FUNCTION_BLOCK MoveVelo IMPLEMENTS I_MoveVelo
VAR
	mcMoveVelo : MC_MoveVelocity;
END_VAR
VAR_IN_OUT
	Axis : AXIS_REF;
END_VAR

mcMoveVelo(Axis := Axis);

PROPERTY Acceleration : MC_LREAL
GET
Acceleration := mcMoveVelo.Acceleration;
END_GET
SET
mcMoveVelo.Acceleration := Acceleration;
END_SET
END_PROPERTY

PROPERTY BufferMode : MC_Buffermode
GET
BufferMode := mcMoveVelo.BufferMode;
END_GET
SET
mcMoveVelo.BufferMode := BufferMode;
END_SET
END_PROPERTY

PROPERTY Busy : BOOL
GET
Busy := mcMoveVelo.Busy;
END_GET
END_PROPERTY

PROPERTY Deceleration : MC_LREAL
GET
Deceleration := mcMoveVelo.Deceleration;
END_GET
SET
mcMoveVelo.Deceleration := Deceleration;
END_SET
END_PROPERTY

PROPERTY Direction : MC_Direction
GET
Direction := mcMoveVelo.Direction;
END_GET
SET
mcMoveVelo.Direction := Direction;
END_SET
END_PROPERTY

PROPERTY Done : BOOL
GET
Done := mcMoveVelo.Done;
END_GET
END_PROPERTY

PROPERTY Error : BOOL
GET
Error := mcMoveVelo.Error;
END_GET
END_PROPERTY

PROPERTY Execute : BOOL
GET
Execute := mcMoveVelo.Execute;
END_GET
SET
mcMoveVelo.Execute := Execute;
END_SET
END_PROPERTY

PROPERTY InVelocity : BOOL
GET
InVelocity := mcMoveVelo.InVelocity;
END_GET
END_PROPERTY

PROPERTY Jerk : MC_LREAL
GET
Jerk := mcMoveVelo.Jerk;
END_GET
SET
mcMoveVelo.Jerk := Jerk;
END_SET
END_PROPERTY

PROPERTY Velocity : MC_LREAL
GET
Velocity := mcMoveVelo.Velocity;
END_GET
SET
mcMoveVelo.Velocity := Velocity;
END_SET
END_PROPERTY

END_FUNCTION_BLOCK

(* stored: Version 1.1.0.1
   POU MoveVelo: Id {11334e21-52f4-414b-aae4-bc02cc7be0a4}, SpecialFunc None
   Property Acceleration: Id {58f1d593-40f0-476d-a5a7-9b3cb778c7d3}
   Get Get: Id {954d0383-4be7-4b14-9478-9d1fb760cc0e}
   Set Set: Id {fc4bfc0a-ae1e-4e71-8268-d6b467dad374}
   Property BufferMode: Id {acef93d6-5f3f-4775-9fbb-a2c1a4097a54}
   Get Get: Id {fc2e896c-3b8e-490c-bad6-bfe7d1ca6171}
   Set Set: Id {3885e3b8-2b10-4b89-92bf-e144af053276}
   Property Busy: Id {316065bc-29d0-4424-a035-e7821cbdb68e}
   Get Get: Id {0304dd71-866f-4d72-94c8-7ce48bc29350}
   Property Deceleration: Id {0eca7112-34e1-452d-bd83-525911101f9b}
   Get Get: Id {9842a6ef-5c35-42d2-8b36-160dd385c854}
   Set Set: Id {17eb47c4-2403-436c-b233-af8799c7bf83}
   Property Direction: Id {9ba30298-b9ce-40be-bb76-1c1bfe193f44}
   Get Get: Id {ebf9023d-0093-478e-99d7-1d330d3aecdb}
   Set Set: Id {61d4010a-ef1e-4749-a1d4-5bf91b8a96a8}
   Property Done: Id {e156641a-9883-416e-a2d0-8afd589f5314}
   Get Get: Id {5fab4201-6235-4c95-afb7-40a863c5ef72}
   Property Error: Id {a4d11270-a859-477d-84e9-ce4a7be77c0d}
   Get Get: Id {c799216e-fed2-4058-a638-99da86f6fb4b}
   Property Execute: Id {b93aeefe-0852-4ad3-b4ec-d3a354d2377d}
   Get Get: Id {67943ec2-2fb6-48b3-9781-80d5d3015933}
   Set Set: Id {1612166f-b6fd-4ab9-8363-73a833cbcaad}
   Property InVelocity: Id {dc4b8849-3347-467f-9440-11f836a20a0a}
   Get Get: Id {84b922be-714a-4add-b495-6fe9876106f2}
   Property Jerk: Id {29e82e07-bb25-4cb8-a634-3e15953f585a}
   Get Get: Id {dc12fddc-bba7-46b4-8e99-ac44cb07ebd2}
   Set Set: Id {59f20c34-b7cf-4332-a972-36e1ff366a22}
   Property Velocity: Id {614f8384-3e4c-46bc-b700-659e0304df72}
   Get Get: Id {7b3c1d0a-7617-4c70-9c46-3129ef99657d}
   Set Set: Id {f71133a2-6dee-46ad-acaa-acf20506d56f} *)
